PROGRAM MAIN
VAR
END_VAR

//MTCPLC();
MOTOR1 ();
MOTOR2 ();

END_PROGRAM

(* stored: Version 1.1.0.1, ProductVersion 3.1.4022.12
   POU MAIN: Id {742caf7b-67de-4474-a314-a5093e649f7c}, SpecialFunc None *)
